// TIA Portal V19 export
DATA_BLOCK "readwrite_hmi_interface"   // DB204
{ S7_Optimized_Access := 'TRUE' }
// stored: AutoNumber false, MemoryReserve 0
   VAR RETAIN
      start : Bool;
      busy : Bool;
      done : Bool;
      drive_error : Bool;
      error : Bool;
      errorID : DWord;
   END_VAR
BEGIN
END_DATA_BLOCK
